FUNCTION_BLOCK PUBLIC PAEScaleVolumetric EXTENDS PAEScaleBase IMPLEMENTS IPAScaleVolumetric
VAR_INPUT
END_VAR
VAR_OUTPUT
END_VAR
VAR
	_ActualRateOfFlow : LREAL;
	_DesiredRateOfFlow : LREAL;
	_PulsePerLiter : LREAL;
END_VAR

{attribute 'monitoring' := 'call'}
//{attribute 'TcRpcEnable'}
PROPERTY PUBLIC ActualRateOfFlow : LREAL
GET // PUBLIC
ActualRateOfFlow := _ActualRateOfFlow;
END_GET
SET // PUBLIC
_ActualRateOfFlow := ActualRateOfFlow;
Root.OnPropertyChangedLReal(THIS^, 74, _ActualRateOfFlow);
END_SET
END_PROPERTY

{attribute 'monitoring' := 'call'}
//{attribute 'TcRpcEnable'}
PROPERTY PUBLIC DesiredRateOfFlow : LREAL
GET // PUBLIC
DesiredRateOfFlow := _DesiredRateOfFlow;
END_GET
SET // PUBLIC
_DesiredRateOfFlow := DesiredRateOfFlow;
Root.OnPropertyChangedLReal(THIS^, 73, _DesiredRateOfFlow);
END_SET
END_PROPERTY

METHOD FB_postinit
VAR_INPUT
	root : IACVariobatch;
END_VAR
SUPER^.FB_postinit(root);
root.OnPropertyChangedLReal(THIS^, 72, _PulsePerLiter);
root.OnPropertyChangedLReal(THIS^, 73, _DesiredRateOfFlow);
root.OnPropertyChangedLReal(THIS^, 74, _ActualRateOfFlow);
END_METHOD

METHOD PUBLIC InvokeSetterLReal
VAR_INPUT
	PropertyID : INT;
	PropertyValue : LREAL;
END_VAR
SUPER^.InvokeSetterLReal(PropertyID, PropertyValue);
CASE PropertyID OF
	72:
		PulsePerLiter := PropertyValue;
	73:
		DesiredRateOfFlow := PropertyValue;
	74:
		ActualRateOfFlow := PropertyValue;
END_CASE
END_METHOD

METHOD OnInitMemory
VAR_INPUT
	root : IACVariobatch;
END_VAR
RegisterProperty(root, 72, GCL.cSizeLREAL); //PulsePerLiter
RegisterProperty(root, 73, GCL.cSizeLREAL); //DesiredRateOfFlow
RegisterProperty(root, 74, GCL.cSizeLREAL); //ActualRateOfFlow
SUPER^.OnInitMemory(root);
END_METHOD

{attribute 'monitoring' := 'call'}
//{attribute 'TcRpcEnable'}
PROPERTY PUBLIC PulsePerLiter : LREAL
GET // PUBLIC
PulsePerLiter := _PulsePerLiter;
END_GET
SET // PUBLIC
_PulsePerLiter := PulsePerLiter;
Root.OnPropertyChangedLReal(THIS^, 72, _PulsePerLiter);
END_SET
END_PROPERTY

END_FUNCTION_BLOCK

(* stored: Version 1.1.0.1, ProductVersion 3.1.4024.6
   POU PAEScaleVolumetric: Id {83836b8a-704f-4eaa-a9ec-a1e64b0b9e24}, SpecialFunc None
   Property ActualRateOfFlow: Id {d8ccbdce-25bd-4256-a88d-b15f8eb2f522}
   Get Get: Id {850aefcc-1410-4db1-a540-959ea5404ef8}
   Set Set: Id {96748b67-23e8-4849-a45f-bd0aaa3067c9}
   Property DesiredRateOfFlow: Id {83692ccd-28d1-481e-83bd-e2f17d57a5c0}
   Get Get: Id {2b6ba631-3c7f-4dfb-991a-312a1c63c762}
   Set Set: Id {7963925c-e7b1-4c26-8ea2-0347e542c038}
   Method FB_postinit: Id {9a5d8845-6b33-48cd-bade-6d6c22c6b8a6}
   Method InvokeSetterLReal: Id {fd8f53b3-37fc-4a60-b3fb-8a16e442e782}
   Method OnInitMemory: Id {329fca44-4fca-4cf1-85af-85838d56b6a3}
   Property PulsePerLiter: Id {d901797c-6a7e-406d-8592-412afddd99f6}
   Get Get: Id {32edcbc3-73a2-4824-b953-fb92fb5d0af5}
   Set Set: Id {afd697c1-e06f-420b-acc5-ce1d147bc005} *)
